(* PLC project Unnamed, Unknown Unnamed 1 *)
(* stored: creationDateTime 2021-04-13T08:37:38, modificationDateTime 2021-04-19T10:13:36 *)

FUNCTION_BLOCK MotionGo
  VAR_INPUT
    ENABLE : BOOL := False;
  END_VAR
  VAR
    SENT : BOOL := False;
  END_VAR
  VAR_OUTPUT
    VALID : BOOL := False;
  END_VAR

            {{
  bool enable = GetFbVar(ENABLE);
  bool sent = GetFbVar(SENT);
  int fd = open("/tmp/MotionGo.pipe",O_RDWR | O_NONBLOCK);
  if(enable && !sent){
    //int fd = open("/tmp/MotionGo.pipe",O_WRONLY | O_NONBLOCK);
    if(fd > 0){
      char buf[1] = {'g'};
      int ret = write(fd, buf, 1);
      if (ret > 0){
        SetFbVar(SENT, true);
      }
    }
  }
  else if(sent){
    //int fd = open("/tmp/MotionGo.pipe",O_RDONLY | O_NONBLOCK);
    char buf[1];
    int ret = read(fd, buf, 1);
    if (ret > 0 && buf[0] == 's'){
      SetFbVar(VALID,true);
    }
  }
  close(fd);
}}
          
END_FUNCTION_BLOCK

PROGRAM program0
  VAR
    LocalVar0 : BOOL := False;
    LocalVar1 : BOOL := False;
    MotionGo0 : MotionGo;
  END_VAR

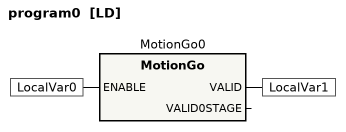
(* LD diagram, written out as Structured Text *)
MotionGo0(ENABLE := LocalVar0);
LocalVar1 := MotionGo0.VALID;
END_PROGRAM

FUNCTION_BLOCK MoveAbsJoint
  VAR_INPUT
    ENABLE : BOOL := False;
  END_VAR
  VAR
    SENT : BOOL := False;
  END_VAR
  VAR_INPUT
    AXIS1 : REAL := 0.0;
    AXIS2 : REAL := 0.0;
    AXIS3 : REAL := 0.0;
    AXIS4 : REAL := 0.0;
    AXIS5 : REAL := 0.0;
    AXIS6 : REAL := 0.0;
    OUTER_AXIS1 : REAL := 0.0;
    OUTER_AXIS2 : REAL := 0.0;
    OUTER_AXIS3 : REAL := 0.0;
    OUTER_AXIS4 : REAL := 0.0;
    OUTER_AXIS5 : REAL := 0.0;
    OUTER_AXIS6 : REAL := 0.0;
    LOAD1 : REAL := 0.0;
    LOAD2 : REAL := 0.0;
    LOAD3 : REAL := 0.0;
    LOAD4 : REAL := 0.0;
    LOAD5 : REAL := 0.0;
    LOAD6 : REAL := 0.0;
    LOAD7 : REAL := 0.0;
    LOAD8 : REAL := 0.0;
    LOAD9 : REAL := 0.0;
    LOAD10 : REAL := 0.0;
    VELOCITY : REAL := 1.0;
    ARC : REAL := 0.0;
  END_VAR
  VAR_OUTPUT
    VALID : BOOL := False;
    ERROR : BOOL := False;
    ERRORID : SINT := 0;
  END_VAR

            {{
  #include <string.h>
  bool enable = GetFbVar(ENABLE);
  bool sent = GetFbVar(SENT);
  if(enable && !sent){
    float axis[6];
    axis[0] = GetFbVar(AXIS1);
    axis[1] = GetFbVar(AXIS2);
    axis[2] = GetFbVar(AXIS3);
    axis[3] = GetFbVar(AXIS4);
    axis[4] = GetFbVar(AXIS5);
    axis[5] = GetFbVar(AXIS6);
    
    float outeraxis[6];
    outeraxis[0] = GetFbVar(AXIS1);
    outeraxis[1] = GetFbVar(AXIS2);
    outeraxis[2] = GetFbVar(AXIS3);
    outeraxis[3] = GetFbVar(AXIS4);
    outeraxis[4] = GetFbVar(AXIS5);
    outeraxis[5] = GetFbVar(AXIS6);
    
    float load[10];
    load[0] = GetFbVar(LOAD1);
    load[1] = GetFbVar(LOAD2);
    load[2] = GetFbVar(LOAD3);
    load[3] = GetFbVar(LOAD4);
    load[4] = GetFbVar(LOAD5);
    load[5] = GetFbVar(LOAD6);
    load[6] = GetFbVar(LOAD7);
    load[7] = GetFbVar(LOAD8);
    load[8] = GetFbVar(LOAD9);
    load[9] = GetFbVar(LOAD10);
    
    float velocity = GetFbVar(VELOCITY);
    float arc = GetFbVar(ARC);
    
    char msg[500]={"MoveAbsJoint,"};
    char word[10];
    
    for(int i=0; i<6; i++){
      sprintf(word, "%.2lf", axis[i]);
      strcat(msg,word);
      strcat(msg,",");
    }
    for(int i=0; i<6; i++){
      sprintf(word, "%.2lf", outeraxis[i]);
      strcat(msg,word);
      strcat(msg,",");
    }
    for(int i=0; i<10; i++){
      sprintf(word, "%.2lf", load[i]);
      strcat(msg,word);
      strcat(msg,",");
    }
    sprintf(word, "%.4lf", velocity);
    strcat(msg,word);
    strcat(msg,",");
    sprintf(word, "%.2lf", arc);
    strcat(msg,word);
    int fd = open("/tmp/MoveAbsJoint.pipe",O_WRONLY | O_NONBLOCK);
    int ret1 = write(fd, msg, 500);
    if (ret1 > 0){
      SetFbVar(SENT,true);
    }
    
  }
  else if(sent){
    //If sent, get result
    int fd = open("/tmp/MoveAbsJoint.pipe",O_RDONLY | O_NONBLOCK);
    char buf[3];
    int ret2 = read(fd, buf, 3);
    if (ret2 > 0){
      if (buf[0] =='y'){
        SetFbVar(VALID, true);
        SetFbVar(ERROR, false);
        SetFbVar(ERRORID, 0);
      }
      else{
        SetFbVar(VALID, false);
        SetFbVar(ERROR, true);
        SetFbVar(ERRORID, buf[1]);
      }
    }
    close(fd);
  } 
  
  
}}
          
END_FUNCTION_BLOCK

FUNCTION_BLOCK GetCurJoint
  VAR_INPUT
    ENABLE : BOOL := False;
  END_VAR
  VAR
    SENT : BOOL := False;
  END_VAR
  VAR_OUTPUT
    VALID : BOOL := False;
    ERROR : BOOL := False;
    ERRORID : SINT := 0;
    AXIS1 : REAL := 0.0;
  END_VAR
  VAR
    AXIS7 : REAL := 0.0;
  END_VAR
  VAR_OUTPUT
    AXIS2 : REAL := 0.0;
    AXIS3 : REAL := 0.0;
    AXIS4 : REAL := 0.0;
    AXIS5 : REAL := 0.0;
    AXIS6 : REAL := 0.0;
  END_VAR
  VAR
    AXIS8 : REAL := 0.0;
  END_VAR

            {{
  #include<string.h>
  bool enable = GetFbVar(ENABLE);
  bool sent = GetFbVar(SENT);
  if(enable && !sent){
    //Send Request
    char buf[1];
    buf[0] = 'g';
    int fd1 = open("/tmp/GetCurJoint.pipe",O_WRONLY | O_NONBLOCK);
    int ret1 = write(fd1, buf, 1);
    if(ret1 > 0){
      SetFbVar(SENT, true);
    }
    close(fd1);
  }
  else if(sent){
    //Get Result
    char buf[100];
    int fd2 = open("/tmp/GetCurJoint.pipe",O_RDONLY | O_NONBLOCK);
    int ret2 = read(fd2, buf, 100);
    if(ret2>0){
      if(buf[0]=='n'){
        //ERROR
        SetFbVar(ERROR, true);
        //1-digit error id
        SetFbVar(ERRORID, buf[1] - 48);
      }
      else if(buf[0] == 'y'){
        //Set Result
        SetFbVar(VALID, true);
        //Set Axises
        char* p;
        int i,j;
        //1
        
        p = strchr(buf, ',');
        i = (int)(p - buf);
        char word[10] = {};
        strncpy(word, buf + 1, i - 1);
        float axis = atof(word);
        SetFbVar(AXIS1, axis);
        SetFbVar(AXIS7, axis);
        //2
        p = strchr(buf + i + 1, ',');
        j = (int)(p - buf);
        strncpy(word, buf + i + 1, j - i -1);
        axis = atof(word);
        SetFbVar(AXIS2, axis);
        i = j;
        //3
        p = strchr(buf + i + 1, ',');
        j = (int)(p - buf);
        strncpy(word, buf + i + 1, j - i - 1);
        axis = atof(word);
        SetFbVar(AXIS3, axis);
        i = j;
        //4
        p = strchr(buf + i + 1, ',');
        j = (int)(p - buf);
        strncpy(word, buf + i + 1, j - i - 1);
        axis = atof(word);
        SetFbVar(AXIS4, axis);
        i = j;
        //5
        p = strchr(buf + i + 1, ',');
        j = (int)(p - buf);
        strncpy(word, buf + i + 1, j - i - 1);
        axis = atof(word);
        SetFbVar(AXIS5, axis);
        i = j;
        //6
        p = strchr(buf + i + 1, ',');
        j = (int)(p - buf);
        strncpy(word, buf + i + 1, j - i - 1);
        axis = atof(word);
        SetFbVar(AXIS6, axis);
        SetFbVar(AXIS8, axis);
        
        
      }
    }
    else{
      //Wait for result
    }
    close(fd2);
  }
  
}}
          
END_FUNCTION_BLOCK

CONFIGURATION Config0
  RESOURCE Res0 ON PLC
    TASK task0(INTERVAL := T#50ms, PRIORITY := 0);
    PROGRAM instance0 WITH task0 : program0;
  END_RESOURCE
END_CONFIGURATION
